{attribute 'linkalways'} 
{attribute 'no_explicit_call' := 'This FB is a CLASS and must be accessed using methods or properties'}
{attribute 'enable_dynamic_creation'}
FUNCTION_BLOCK Node_F_VN_FillContainer_UINT EXTENDS VisionNode
VAR
    ipContainer : _ITcVnContainer;
    nValue : _UINT(0);
    hrPrev : _HRESULT(S_OK);
    hresult : _HRESULT(S_OK);
END_VAR

METHOD PUBLIC  Clone : I_Node
VAR
    pNode : POINTER TO Node_F_VN_FillContainer_UINT;
END_VAR
pNode := __NEW(Node_F_VN_FillContainer_UINT);
Clone := pNode^;
END_METHOD

METHOD FB_init : BOOL
VAR_INPUT
    bInitRetains : BOOL; // if TRUE, the retain variables are initialized (warm start / cold start)
    bInCopyCode : BOOL;  // if TRUE, the instance afterwards gets moved into the copy code (online change)
END_VAR
AddInput('ipContainer', ipContainer);
AddParameter('nValue', nValue);
AddInput('hrPrev', hrPrev);
AddOutput('ipContainer', ipContainer);
AddOutput('hresult',hresult);
END_METHOD

METHOD PROTECTED OnExecute
hresult.Value := F_VN_FillContainer_UINT(
    ipContainer := ipContainer.Value,
    nValue := nValue.Value,
    hrPrev:= hrPrev.Value);
END_METHOD

METHOD PUBLIC PreExecutionCheck
VAR_INPUT
    Check : I_PreExecutionChecks;
END_VAR
Check.IsTrue(ipContainer.IsValid, 'ipContainer must be a valid container');
Check.IsTrue(ipContainer.IsType(TC_GLOBAL_CONST_LIST.ContainerType_Vector_UINT), 'ipContainer contains incorrect type');
END_METHOD

END_FUNCTION_BLOCK

(* stored: Version 1.1.0.1, ProductVersion 3.1.4026.13
   POU Node_F_VN_FillContainer_UINT: Id {4972972f-8397-4242-b6ff-e33ae8b4941e}, SpecialFunc None
   Folder Constructor: Id {e5744687-9b4e-45a6-b833-d4ae9db9819f}
   Method Clone: Id {66b4198e-96fd-4ae3-ba85-e425380442ee}
   Method FB_init: Id {c31c5664-d91a-4883-acd4-fd4bd4c76eb7}
   Method OnExecute: Id {b4a507d6-1cc2-4917-adaf-60a012a79c35}
   Method PreExecutionCheck: Id {29556564-4d94-49db-81d1-d7c246cd0ae5} *)
